FUNCTION_BLOCK SchieberVerriegelungComposite (* Composite FB wrapping other FBs *)
  (* Standard: 61499-2; Description: Copyright (c) 2025 HR Agrartechnik GmbH This program and the accompanying materials are made available under the terms of the Eclipse Public License 2.0 which is available at https://www.eclipse.org/legal/epl-2.0/ SPDX-License-Identifier: EPL-2.0 *)
  (* Version 1.0, 2025-06-04, Franz Höpfinger, HR Agrartechnik GmbH *)
  PACKAGE logiBUS::utils::sequence::schieber;
  IMPORT eclipse4diac::core::TypeHash;
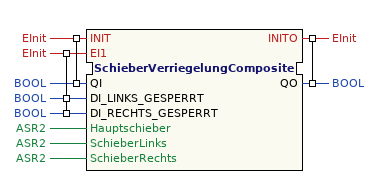
  EVENT_INPUT
    INIT : EInit WITH QI; (* Initialization Request *)
    EI1 : EInit WITH DI_LINKS_GESPERRT, DI_RECHTS_GESPERRT;
  END_EVENT
  EVENT_OUTPUT
    INITO : EInit WITH QO; (* Initialization Confirm *)
  END_EVENT
  VAR_INPUT
    QI : BOOL; (* Input event qualifier *)
    DI_LINKS_GESPERRT : BOOL;
    DI_RECHTS_GESPERRT : BOOL;
  END_VAR
  VAR_OUTPUT
    QO : BOOL; (* Output event qualifier *)
  END_VAR
  SOCKETS
    Hauptschieber : adapter::types::bidirectional::ASR2;
    SchieberLinks : adapter::types::bidirectional::ASR2;
    SchieberRechts : adapter::types::bidirectional::ASR2;
  END_SOCKETS
  FBS
    SchieberVerriegelung : logiBUS::utils::sequence::schieber::SchieberVerriegelung;
  END_FBS
  EVENT_CONNECTIONS
    INIT TO SchieberVerriegelung.INIT;
    SchieberVerriegelung.INITO TO INITO;
    Hauptschieber.EO_SET TO SchieberVerriegelung.EI_Hauptschieber_Open;
    Hauptschieber.EO_RESET TO SchieberVerriegelung.EI_Hauptschieber_Close;
    SchieberRechts.EO_SET TO SchieberVerriegelung.EI_SchieberRechts_Open;
    SchieberRechts.EO_RESET TO SchieberVerriegelung.EI_SchieberRechts_Close;
    SchieberLinks.EO_SET TO SchieberVerriegelung.EI_SchieberLinks_Open;
    SchieberLinks.EO_RESET TO SchieberVerriegelung.EI_SchieberLinks_Close;
    SchieberVerriegelung.EO_Hauptschieber_Open TO Hauptschieber.EI_SET;
    SchieberVerriegelung.EO_Hauptschieber_Close TO Hauptschieber.EI_RESET;
    SchieberVerriegelung.EO_SchieberLinks_Open TO SchieberLinks.EI_SET;
    SchieberVerriegelung.EO_SchieberLinks_Close TO SchieberLinks.EI_RESET;
    SchieberVerriegelung.EO_SchieberRechts_Open TO SchieberRechts.EI_SET;
    SchieberVerriegelung.EO_SchieberRechts_Close TO SchieberRechts.EI_RESET;
    EI1 TO SchieberVerriegelung.EI1;
  END_CONNECTIONS
  DATA_CONNECTIONS
    QI TO SchieberVerriegelung.QI;
    SchieberVerriegelung.QO TO QO;
    DI_LINKS_GESPERRT TO SchieberVerriegelung.DI_LINKS_GESPERRT;
    DI_RECHTS_GESPERRT TO SchieberVerriegelung.DI_RECHTS_GESPERRT;
  END_CONNECTIONS
END_FUNCTION_BLOCK
